// TIA Portal V19 export
DATA_BLOCK "PPrgArchive19"   // DB515
// stored: IsOnlyStoredInLoadMemory true, MemoryReserve 0, Namespace G
   VAR RETAIN
      PRG : Array[1801..1900] of "PPrg_Data";
   END_VAR
BEGIN
END_DATA_BLOCK
